// TIA Portal V17 export
// export: Created 2024-09-02T12:50:27.1956498Z, ExportSetting WithDefaults, DisplayName Totally Integrated Automation Portal, DisplayVersion V17, DisplayName TIA Portal Openness, DisplayVersion V17, DisplayName TIA Portal Version Control Interface, DisplayVersion V17, DisplayName STEP 7 Professional, DisplayVersion V17, DisplayName STEP 7 Safety, DisplayVersion V17, DisplayName WinCC Professional, DisplayVersion V17
TYPE "TypeStepsHand"
// stored: IsFailsafeCompliant false
   STRUCT
      INIT : Bool := true;
      INIT_HM_fp : Bool;
      Ready_SYS_INIT_HMI : Bool;
      Z : Array[1..348] of Struct
         Pair_Error : Bool;   // Paarfehler vorhanden / Pair error present
         Pair_Error_Timer { S7_SetPoint := 'True'} : TON_TIME;
         dbInstanceName { S7_SetPoint := 'True'} : WString[125];
         stepNumber_Left : USInt;
         stepNumber_Right : USInt;
      END_STRUCT;
   END_STRUCT;
END_TYPE
